FUNCTION_BLOCK E_MERGE_4 (* Basic Function Block Type *)
  (* Standard: 61499-2 *)
  (* Version 0.0, 2/4/2026, SESA713705, Schneider Electric, Template *)
  PACKAGE SE.Nereda;
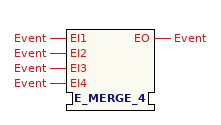
  EVENT_INPUT
    EI1;
    EI2;
    EI3;
    EI4;
  END_EVENT
  EVENT_OUTPUT
    EO;
  END_EVENT
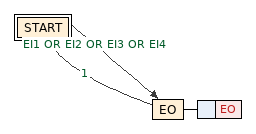
  EC_STATES
    START; (* Initial State *)
    EO : -> EO;
  END_STATES
  EC_TRANSITIONS
    START TO EO := EI1 OR EI2 OR EI3 OR EI4;
    EO TO START := 1;
  END_TRANSITIONS
END_FUNCTION_BLOCK
